(* PLC project Substation_Feeder_Automation_Controls.project, CODESYS CODESYS V3.5 SP22 Patch 3 *)
(* stored: creationDateTime 2026-09-24T12:18:53.7208919, modificationDateTime 2026-09-24T11:11:14.0125883 *)

PROGRAM PLC_PRG
VAR



    {attribute 'symbol' := 'readwrite'}
    Mode_Remote             : BOOL := TRUE;
    {attribute 'symbol' := 'readwrite'}
    Sts_DC_Healthy          : BOOL := TRUE;
    {attribute 'symbol' := 'readwrite'}
    Sts_Protection_Healthy  : BOOL := TRUE;
    {attribute 'symbol' := 'readwrite'}
    Sts_CB_Open             : BOOL := TRUE;
    {attribute 'symbol' := 'readwrite'}
    Sts_BusDS_Closed        : BOOL := TRUE;
    {attribute 'symbol' := 'readwrite'}
    Sts_LineDS_Closed       : BOOL := TRUE;
    {attribute 'symbol' := 'readwrite'}
    Sts_GroundDS_Open       : BOOL := TRUE;
    {attribute 'symbol' := 'readwrite'}
    Sts_Lockout86           : BOOL := FALSE;

    {attribute 'symbol' := 'read'}
    Perm_CB_Close           : BOOL := FALSE;
    {attribute 'symbol' := 'read'}
    Out_CB_Close            : BOOL := FALSE;
    {attribute 'symbol' := 'read'}
    Out_CB_Open             : BOOL := FALSE;
END_VAR
VAR_INPUT
    {attribute 'symbol' := 'readwrite'}
	Cmd_CB_Close            : BOOL := FALSE;
    {attribute 'symbol' := 'readwrite'}
    Cmd_CB_Open             : BOOL := FALSE;
END_VAR

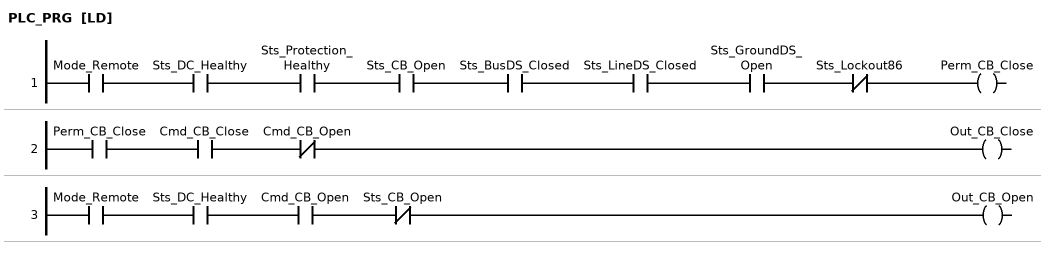
(* LD diagram, written out as Structured Text *)
(* Close permissive: all isolator, protection, DC and remote-mode conditions healthy; no 86 lockout. *)

Perm_CB_Close := Mode_Remote AND Sts_DC_Healthy AND Sts_Protection_Healthy AND Sts_CB_Open AND Sts_BusDS_Closed AND Sts_LineDS_Closed AND Sts_GroundDS_Open AND NOT Sts_Lockout86;
(* Close output: valid permissive and close request. Open request always inhibits close. *)

Out_CB_Close := Perm_CB_Close AND Cmd_CB_Close AND NOT Cmd_CB_Open;
(* Remote open output: DC healthy and breaker not already open. Close-only interlocks do not block opening. *)

Out_CB_Open := Mode_Remote AND Sts_DC_Healthy AND Cmd_CB_Open AND NOT Sts_CB_Open;
END_PROGRAM

PROGRAM Heartbeat
VAR
    {attribute 'symbol' := 'read'}
    Counter : UDINT := 0;
    PulseTimer : TON;
    CommandTimer : TON;
END_VAR

            // Called after PLC_PRG in the same MainTask.
// Increment every ~500 ms. Explicit wrap avoids overflow exceptions.
PulseTimer(IN := NOT PulseTimer.Q, PT := T#500ms);
IF PulseTimer.Q THEN
    IF Counter >= UDINT#4294967295 THEN
        Counter := 0;
    ELSE
        Counter := Counter + 1;
    END_IF;
END_IF;

// Lab HMI command duration guard. This POU runs after PLC_PRG.
// Independent of browser/Gateway cleanup; outputs recompute next 20 ms scan.
CommandTimer(IN := PLC_PRG.Cmd_CB_Open OR PLC_PRG.Cmd_CB_Close, PT := T#7s);
IF CommandTimer.Q THEN
    PLC_PRG.Cmd_CB_Open := FALSE;
    PLC_PRG.Cmd_CB_Close := FALSE;
END_IF;

          
END_PROGRAM
